FUNCTION_BLOCK FB_DerotatorControl EXTENDS FB_AxisControl
VAR_INPUT
END_VAR
VAR_OUTPUT
END_VAR
VAR
	tonTorqueError		: TON := (PT := T#3S);	// trigger for the torque error
END_VAR

(*
Selection 6
Homing in Endlage:

https://infosys.beckhoff.com/index.php?content=../content/1031/ax5000_usermanual/html/ax5000_homing_hardware_end_position.htm&id=12221
NC-Interface:
PlcToNc-Achsinterface, Bit 8 namens AcceptBlockedDriveSignal im nDeCtrlDWord

SPS-Interface:
TcNc-Lib, siehe SPS-Funktion AxisSetAcceptBlockedDriveSignal in der TwinCAT  PLC Library: NC.
*)

fPosition := LIMIT(fMinPosition, fPosition, fMaxPosition);

IF bEnable AND NOT fbAxis.Calibrated THEN
	bHomeAxis := TRUE;
END_IF

IF fbAxis.Calibrated THEN
	bHomeAxis := FALSE;
	bCalibrated := fbAxis.Calibrated;
END_IF
	
IF bHomeAxis THEN
	fPosition := fCalibPosition;
END_IF

fbAxis(
	enable 			:= bEnable,
	Reset 			:= bReset,
	MoveAxis 		:= bMoveAxis,
	HomeAxis 		:= bHomeAxis,
	StopAxis 		:= bStopAxis,
	HomingMode 		:= MC_ForceCalibration,
	Position 		:= fPosition, 
	Velocity 		:= fVelocity,
	Enable_Positive := TRUE,
	Enable_Negative := TRUE,
	Jog_Forward 	:= bMovePos,
	Jog_Backwards 	:= bMoveNeg,
	bCalibrationCam := inDigitalInputs.0,
	isModuloAxis 	:= FALSE,
	Tracking 		:= bTracking,
	ActualPosition 	=> fActualPosition,
	Error 			=> bError,
	ErrorID 		=> nErrorID,
	AxisRef 		:= axisRef);
	
IF fbAxis.MoveDone OR bReset OR bError THEN
	bMoveAxis := FALSE;
END_IF

IF fbAxis.HomeDone OR bReset OR bError THEN
	bHomeAxis := FALSE;
END_IF
	
IF fbAxis.ResetDone THEN
	bReset := FALSE;
END_IF

IF fbAxis.StopDone THEN
	bStopAxis := FALSE;
END_IF

bDiagnosticError := FALSE;
IF inDiagnostic < 16#D012 AND inDiagnostic > 16#D014 THEN
	bDiagnosticError := TRUE;
	nErrorID := inDiagnostic;
	bSoeReset := bReset;
END_IF

bReady := fbAxis.Ready;

fbReadParameter(	
	Axis 			:= axisRef, 
	Enable 			:= fbAxis.InMotion, 
	ParameterNumber := MC_AxisParameter.AxisRemainingTimeToGo, 
	ReadMode 		:= E_ReadMode.READMODE_CYCLIC);
				
IF fbReadParameter.Valid THEN
	fSlewTime := fbReadParameter.Value;
END_IF

IF bSoEReset THEN
	fbSoEReset(
		Axis 	:= axisRef,
		Execute := TRUE,
		Timeout := DEFAULT_ADS_TIMEOUT);
 	IF NOT fbSoEReset.Busy THEN
		fbSoEReset(Axis := axisRef, Execute := FALSE);
		bSoEReset := FALSE;
		bReset := TRUE;
	END_IF
END_IF

fTorque := inTorque / 10.0;
// nominal torque is 3%, max is 25%
tonTorqueError(IN := ABS(fTorque) > 20.0);

axisEvent(	
	Trigger 		:= bError, 
	Level 			:= ADSLOG_MSGTYPE_ERROR,
	FormatString	:= 'Derotator Axis Error: %s',
	OnMessage 		:= NCError_TO_STRING(nErrorID),
	OffMEssage 		:= 'OK',
	OffLevel 		:= ADSLOG_MSGTYPE_HINT,
	Comm			:= fbComm);
	
diagnosticEvent(	
	Trigger 		:= bDiagnosticError, 
	Level 			:= ADSLOG_MSGTYPE_ERROR,
	FormatString	:= 'Derotator Axis Diagnostic Error: %s',
	OnMessage 		:= NCError_TO_STRING(inDiagnostic),
	Comm			:= fbComm);
	
TorqueWarning(	
	Trigger 		:= tonTorqueError.Q, 
	Level 			:= ADSLOG_MSGTYPE_WARN,
	FormatString 	:= '%s',
	OnMessage 		:= 'Derotator torque is high.',
	Comm			:= fbComm);

CalibrationEvent(	
	Trigger 		:= bCalibrated, 
	Level 			:= ADSLOG_MSGTYPE_HINT,
	OnMessage 		:= 'Derotator is calibrated.',
	Comm			:= fbComm);

PROPERTY InNegLimit : BOOL
GET
InNegLimit := inDigitalInputs.1;
END_GET
END_PROPERTY

PROPERTY InPosLimit : BOOL
GET
InPosLimit := inDigitalInputs.0;
END_GET
END_PROPERTY

END_FUNCTION_BLOCK

(* stored: Version 1.1.0.1, ProductVersion 3.1.4024.15
   POU FB_DerotatorControl: Id {acfc3cc1-a4bd-4873-ba58-50b0c54d8bf5}, SpecialFunc None
   Property InNegLimit: Id {5e7f9e66-b876-444b-bc02-75ea47096cf0}
   Get Get: Id {2b9866db-9dc6-47f0-beb6-6e3aa86d150c}
   Property InPosLimit: Id {a6e23b26-e079-44fd-b036-d5b41f19b37a}
   Get Get: Id {da8f7515-fc44-4a5a-a8b6-b5f4a39e4ba6} *)
